// Read-only view of the configured EtherCAT slaves, indexed 0-based in configuration order.
// EtherCatMaster implements it; SyncUnitTask and other collaborators that only need to resolve
// slaves depend on this contract instead of on the whole master.
INTERFACE I_EcSlaveRegistry EXTENDS I_Base

{attribute 'monitoring' := 'call'}
PROPERTY ConfiguredSlaveCount : UINT
GET
END_GET
END_PROPERTY

// Configured slave index (0-based) of the slave with EtherCAT address Addr, -1 if none.
// O(1) for the dense address range starting at 1001, linear search otherwise.
METHOD GetSlaveIndexByAddr : DINT
VAR_INPUT
	Addr : UINT;
END_VAR
END_METHOD

// Name of the configured slave at Index, '' if Index is out of range.
METHOD GetSlaveName : STRING
VAR_INPUT
	Index : UINT;
END_VAR
END_METHOD

// TRUE if the configured slave at Index belongs to a hot connect group (topology status bits 4 or 5).
// FALSE if Index is out of range.
METHOD IsHotConnectMember : BOOL
VAR_INPUT
	Index : UINT;
END_VAR
END_METHOD

END_INTERFACE

(* stored: Version 1.1.0.1, ProductVersion 3.1.4026.27
   Itf I_EcSlaveRegistry: Id {7ecd9ba6-d0e2-4c1f-ab63-8e024170d7f5}
   Property ConfiguredSlaveCount: Id {69b8a77d-8601-4098-bed0-bb5963e01edb}
   Get Get: Id {e9dc7296-1fcc-4ef5-a9ab-99fef2c652e0}
   Method GetSlaveIndexByAddr: Id {fe76d2a1-904b-493d-b227-045ce9d15c25}
   Method GetSlaveName: Id {f0578778-594b-4c69-aab7-c0ed3eaa0640}
   Method IsHotConnectMember: Id {1381a31c-5c4f-4c2b-a5f6-b00af3f5750c} *)
